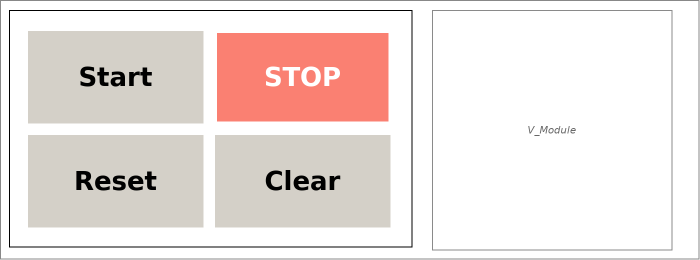
VISUALIZATION V_MachineModule  // 700x260
VAR_IN_OUT
	HMI : ST_PackMLBaseModule_HMI;
END_VAR
    Frame (432,10 240x240)
        shows V_Module(HMI := HMI)
    RoundedRectangle (9,10 403x237)
    RoundedRectangle (28,31 175x92), "Start"
        OnMouseClick: execute { HMI.Command.State := E_PMLCommand.ePMLCommand_Start; }
    RoundedRectangle (215,135 175x92), "Clear"
        OnMouseClick: execute { HMI.Command.State := E_PMLCommand.ePMLCommand_Clear; }
    RoundedRectangle (28,135 175x92), "Reset"
        OnMouseClick: execute { HMI.Command.State := E_PMLCommand.ePMLCommand_Reset; }
    RoundedRectangle (215,31 175x92), "STOP"
        toggle SafetyGlobalVariableList.eStopHMI
        OnMouseClick: execute {  }
END_VISUALIZATION

(* stored: Version 1.1.0.1, ProductVersion 3.1.4024.15
   Visu V_MachineModule: Id {36f6a3ae-b99e-0ef0-3759-f9efb58a3c39} *)
